{attribute 'linkalways'} 
{attribute 'no_explicit_call' := 'This FB is a CLASS and must be accessed using methods or properties'}
{attribute 'enable_dynamic_creation'}
FUNCTION_BLOCK FINAL MAX_USINT EXTENDS Node
VAR
	in1 : _USINT(0);
	in2 : _USINT(0);
	out : _USINT(0);
END_VAR

METHOD PUBLIC Clone : I_Node
VAR
	pNode : POINTER TO MAX_USINT;
END_VAR
pNode := __NEW(MAX_USINT);
Clone := pNode^;
END_METHOD

METHOD FB_init : BOOL
VAR_INPUT
	bInitRetains : BOOL; // if TRUE, the retain variables are initialized (warm start / cold start)
	bInCopyCode : BOOL;  // if TRUE, the instance afterwards gets moved into the copy code (online change)
END_VAR
AddInput('in1',THIS^.in1);
AddInput('in2',THIS^.in2);
AddOutput('out', THIS^.out);
END_METHOD

METHOD PROTECTED OnExecute
VAR
END_VAR
out.Value := MAX(in1.Value, in2.Value);
END_METHOD

END_FUNCTION_BLOCK

(* stored: Version 1.1.0.1, ProductVersion 3.1.4024.15
   POU MAX_USINT: Id {2b8b0195-1f1f-4cf0-9368-08b6403a8b5d}, SpecialFunc None
   Folder Constructor: Id {1bf1ba44-e143-40dd-b147-156a1c7fa5ee}
   Method Clone: Id {67b19d5b-ab29-4e22-ae3b-8ac1fb08bba8}
   Method FB_init: Id {3dd18088-e992-4d17-abb4-6dc0c1bdb158}
   Method OnExecute: Id {aaa37bb3-cf59-4f20-96a6-826f6e3aa3b7} *)
